INTERFACE I_Interface

END_INTERFACE

(* stored: Version 1.1.0.1, ProductVersion 3.1.4024.12
   Itf I_Interface: Id {7a6c06c8-6b80-4a13-b850-ab251192df1e} *)
